Universal Robots URScript: external_control.script

def external_control():
  global _hidden_verificationVariable=0
  set_standard_analog_input_domain(0, 1)
  set_standard_analog_input_domain(1, 1)
  set_tool_analog_input_domain(0, 1)
  set_tool_analog_input_domain(1, 1)
  set_analog_outputdomain(0, 0)
  set_analog_outputdomain(1, 0)
  set_input_actions_to_default()
  set_tool_communication(False, 115200, 0, 1, 1.5, 3.5)
  set_tool_output_mode(0)
  set_tool_digital_output_mode(0, 1)
  set_tool_digital_output_mode(1, 1)
  set_tool_voltage(0)
  set_tcp(p[0.0,0.0,0.0,0.0,0.0,0.0])
  set_target_payload(0.500000, [0.000000, 0.000000, 0.000000], [0.000485, 0.000485, 0.000485, 0.000000, 0.000000, 0.000000])
  set_safety_mode_transition_hardness(1)
  set_gravity([0.0, 0.0, 9.82])
  # begin: URCap Installation Node
  #   Source: External Control, 1.0.5, FZI Research Center for Information Technology
  #   Type: External Control
  # end: URCap Installation Node
  step_count_e23f2d63_c93a_44c0_a6ac_b73dd2b161e3 = 0.0
  thread Step_Counter_Thread_8451ef99_b206_499f_a717_e17b49c67c18():
    while (True):
      step_count_e23f2d63_c93a_44c0_a6ac_b73dd2b161e3 = step_count_e23f2d63_c93a_44c0_a6ac_b73dd2b161e3 + 1.0
      sync()
    end
  end
  run Step_Counter_Thread_8451ef99_b206_499f_a717_e17b49c67c18()
  while (True):
    $ 2 "Robot Program"
    # begin: URCap Program Node
    #   Source: External Control, 1.0.5, FZI Research Center for Information Technology
    #   Type: External Control
    $ 3 "Control by 192.168.12.12"
popup("The connection to the remote PC at 192.168.12.12:50002 could not be established. Reason: Connection refused (Connection refused)","Receive program failed", False, True, blocking=True)
sync()    # end: URCap Program Node
  end
end
